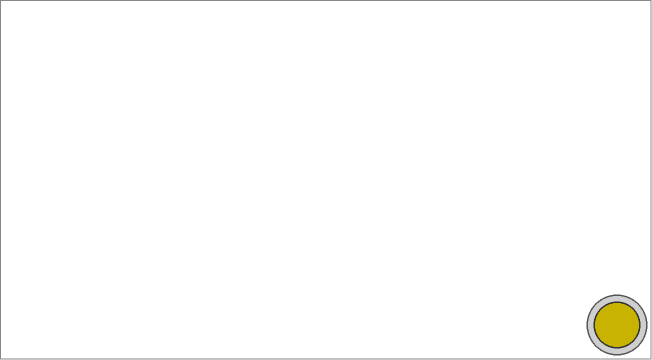
VISUALIZATION Visu  // 652x360
    Lamp1 (582,290 70x70), variable: MAIN.bLamp, style: Lamp-Lamp1-Yellow
END_VISUALIZATION

(* stored: Version 1.1.0.1, ProductVersion 3.1.4024.12
   Visu Visu: Id {b70498bf-8da6-4f84-b5be-063c8cf1b78c} *)
